FUNCTION_BLOCK FD_ConvoyerDevice EXTENDS FD_Device IMPLEMENTS ITF_Convoyer
VAR_INPUT
END_VAR

VAR_OUTPUT
END_VAR

VAR 
	//===================== Variable
	eSource 						 : E_Convoyer;
  eDestination 				 : E_Convoyer;
	
	bRouteRequest				 : BOOL;
	bCarrierWaiting   	 : BOOL;
	bRouteGranted 			 : BOOL;
	
	bTranspOutRequest    : BOOL;
	bTranspOutBusy       : BOOL;
	bTranspOutDone       : BOOL;
	
	//===================== Instance
	fbStopperCarrieConvoyer						: FB_PneuCyl_Stopper  (GVL_Customer.C_Name_StopperCarrieConvoyer,
																													GVL_Customer.C_ID_StopperCarrieConvoyer
																										  		);																												
																												
	fbMotorConvoyer										: FB_SimpleMotor      (GVL_Customer.C_Name_ConvoyerDcMotor,
																													 GVL_Customer.C_ID_MotorComvoyer
																										  		);
																													
	fbReadHead												: FB_ReadHead        	(GVL_Customer.C_Name_ReadHead,
																													GVL_Customer.C_ID_ReadHead
																										  		); 
																													
END_VAR

VAR CONSTANT
	// --------------------------Base------------------
	C_SeqStep_OnBasePos_Start															: UINT :=  1; 
	C_SeqStep_OnBasePos_WaitOpMode												: UINT :=  2;
	C_SeqStep_OnBasePos_Done															: UINT :=  30; 
	
	// --------------------------Auto Sequence------------------
	C_SeqStep_Auto_Start																	: UINT :=  10;
	C_SeqStep_Auto_Wait_Carrier_At_Stopper								: UINT :=  110;
	C_SeqStep_Auto_Read_Destination_Once									: UINT :=  120;
	C_SeqStep_Auto_Ask_RouteManager_For_A_Route						: UINT :=  130;
	C_SeqStep_Auto_Inject_Carrier_IntoGranted_Route				: UINT :=  140;
	C_SeqStep_Auto_End																		: UINT :=  150;
	
END_VAR


//******* Important and necessary
SUPER^();  
//====================================
IF NOT Enable THEN RETURN; END_IF

fbStopperCarrieConvoyer();
fbMotorConvoyer();
fbReadHead();

PROPERTY CarrierWaiting : BOOL
GET
CarrierWaiting := bCarrierWaiting;
END_GET
SET
bCarrierWaiting := CarrierWaiting;
END_SET
END_PROPERTY

PROPERTY Destination : E_Convoyer
GET
Destination := eDestination;
END_GET
SET
eDestination := Destination;
END_SET
END_PROPERTY

//FB_Init ist immer implizit verfügbar und wird primär für die Initialisierung verwendet.
//Der Rückgabewert wird nicht ausgewertet. Für gezielte Einflussnahme können Sie
//die Methoden explizit deklarieren und darin mit dem Standard-Initialisierungscode 
//zusätzlichen Code bereitstellen. Sie können den Rückgabewert auswerten.
METHOD FB_Init: BOOL
VAR_INPUT    
	bInitRetains					: BOOL; 					// TRUE: Die Retain-Variablen werden initialisiert (Reset warm / Reset kalt)    
	bInCopyCode						: BOOL;  					// TRUE: Die Instanz wird danach in den Kopiercode kopiert (Online-Change)
	
	I_Name                : STRING;         //  Name
	I_ID                  : UINT;           // ID
  I_itfOwner					  : ITF_Owner;      // owner 
END_VAR
END_METHOD

METHOD mAutomatic : E_CmdState
VAR_INPUT
	I_bExecute	: BOOL;
END_VAR

SUPER^.mAutomatic(TRUE);
END_METHOD

METHOD mCmdExec_Auto : E_CmdState
VAR_INPUT
END_VAR

VAR
    L_eCmd 			: E_CmdState;
END_VAR

CASE SequenceID OF

  //******************************************************* Idle 
  C_SeqStep_Idle: 
  	SequenceID       :=  C_SeqStep_Start;
  
  //****************************************************** Start
  C_SeqStep_Start:
		bRouteRequest 			:= FALSE;
    bRouteGranted 			:= FALSE;
    bTranspOutRequest 	:= FALSE;
    bTranspOutDone 			:= FALSE; 	
  	SequenceID          := C_SeqStep_Auto_Wait_Carrier_At_Stopper;
		
	C_SeqStep_Auto_Wait_Carrier_At_Stopper :
	
	IF fbStopperCarrieConvoyer.CarriePresent 
		THEN
      SequenceID := C_SeqStep_Auto_Read_Destination_Once;
  END_IF
	
	C_SeqStep_Auto_Read_Destination_Once:
	// Read destination one.
  	IF fbReadHead.mRead(TRUE) = E_CmdState.Succeeded 
			THEN
  	    eDestination 		:= fbReadHead.ReadDestination;
  	    SequenceID 			:= C_SeqStep_Auto_Ask_RouteManager_For_A_Route;
  	END_IF
	
	C_SeqStep_Auto_Ask_RouteManager_For_A_Route:
	// Ask RouteManager for a route.
 		bRouteRequest := TRUE;
		
    IF bRouteGranted 
			THEN
    		bTranspOutRequest  := TRUE;
    	  SequenceID         := C_SeqStep_Auto_Inject_Carrier_IntoGranted_Route;
    	END_IF

	 C_SeqStep_Auto_Inject_Carrier_IntoGranted_Route:
      // Inject carrier into granted route.				
		IF mCmdExec_TranspOut(bTranspOutRequest ) = E_CmdState.Succeeded 
			THEN
      	bRouteRequest     := FALSE;
      	bRouteGranted     := FALSE;
      	bTranspOutRequest := FALSE;
      	SequenceID        := C_SeqStep_Auto_End;
     END_IF
									
  C_SeqStep_Error: 
    //************* all FB reset
 
 	C_SeqStep_Auto_End:
	  //**********************End 
		SequenceID := C_SeqStep_Start;
  		
END_CASE
END_METHOD

METHOD mCmdExec_BasePos : E_CmdState
VAR_INPUT
END_VAR

CASE SequenceID OF
  //******************************************************* Idle 
  C_SeqStep_Idle: 
  	;
  //****************************************************** Start
  C_SeqStep_OnBasePos_Start:
	// Home position for LTU is MIDDLE.
		fbMotorConvoyer.mStopMotor(TRUE);
		IF E_CmdState.Succeeded  = fbStopperCarrieConvoyer.mCallBase(TRUE)
			THEN
				Homed := TRUE;
  	  	Ready := TRUE;
  	  	SequenceID := C_SeqStep_OnBasePos_Done;
		END_IF
		
  C_SeqStep_Error: 
    //************* all FB reset
    mCmdExec_BasePos := mDone(); 
  //**********************Done
 	C_SeqStep_OnBasePos_Done:
  	mCmdExec_BasePos := mDone();
END_CASE
END_METHOD

METHOD mCmdExec_Service : E_CmdState
VAR_INPUT
END_VAR
;
END_METHOD

METHOD mCmdExec_TranspOut : E_CmdState
VAR_INPUT
	I_bExecute 			: BOOL;
END_VAR

IF NOT I_bExecute 
	THEN
    bTranspOutBusy := FALSE;
    mCmdExec_TranspOut := E_CmdState.Idle;
    RETURN;
END_IF

// Route not granted yet.
// Route noch nicht freigegeben
IF NOT bRouteGranted 
	THEN
  	mCmdExec_TranspOut := E_CmdState.NotReady;
    RETURN;
END_IF

bTranspOutBusy := TRUE;
bTranspOutDone := FALSE;

// Open stopper: stopper down = carrier can pass.
fbStopperCarrieConvoyer.mCallWork(TRUE);

// Start conveyor motor.
fbMotorConvoyer.mStartMotor(TRUE);

// Wait until carrier leaves stopper sensor.
IF NOT fbStopperCarrieConvoyer.CarriePresent 
	THEN
  	// Stop local injection.
  	fbMotorConvoyer.mStopMotor(TRUE);
		
  	// Close stopper again.
  	fbStopperCarrieConvoyer.mCallBase(TRUE);
  	bTranspOutBusy := FALSE;
  	bTranspOutDone := TRUE;
  	mCmdExec_TranspOut := E_CmdState.Succeeded;
  	RETURN;
END_IF
END_METHOD

METHOD mHold : E_CmdState
VAR_INPUT
	I_bExecute	: BOOL;
END_VAR
END_METHOD

METHOD mHome : E_CmdState
VAR_INPUT
	I_bExecute	: BOOL;
END_VAR
SUPER^.mHome(I_bExecute);
END_METHOD

METHOD mRelease : E_CmdState
VAR_INPUT
	I_bExecute	: BOOL;
END_VAR
END_METHOD

METHOD mSequence : E_CmdState
VAR_INPUT
	I_bExecute				: BOOL;
END_VAR

VAR
	L_eState 					: E_CmdState;
END_VAR
mSequence := SUPER^.mSequence(I_bExecute);	


// Generic checks from parent
L_eState := SUPER^.mSequence(I_bExecute := I_bExecute);

IF L_eState <> E_CmdState.Busy 
	THEN
    mSequence := L_eState;
    RETURN;
END_IF

CASE Mode OF
	E_Mode.Homing:
		mSequence := mCmdExec_BasePos();
	E_Mode.Auto:
		mSequence := mCmdExec_Auto();
	E_Mode.Service:
		mSequence := mCmdExec_Service();	
END_CASE
END_METHOD

METHOD mService : E_CmdState
VAR_INPUT
	I_bExecute	: BOOL;
END_VAR
END_METHOD

METHOD mStop : E_CmdState
VAR_INPUT
	I_bExecute	: BOOL;
END_VAR
END_METHOD

PROPERTY RouteGranted : BOOL
GET
RouteGranted := bRouteGranted;
END_GET
SET
bRouteGranted := RouteGranted;
END_SET
END_PROPERTY

PROPERTY RouteRequest : BOOL
GET
RouteRequest := bRouteRequest;
END_GET
SET
bRouteRequest := RouteRequest;
END_SET
END_PROPERTY

PROPERTY Source : E_Convoyer
GET
Source := eSource;
END_GET
SET
eSource := Source;
END_SET
END_PROPERTY

PROPERTY TranspOutBusy : BOOL
GET
TranspOutBusy := bTranspOutBusy;
END_GET
SET
bTranspOutBusy := TranspOutBusy;
END_SET
END_PROPERTY

PROPERTY TranspOutDone : BOOL
GET
TranspOutDone := bTranspOutDone;
END_GET
SET
bTranspOutDone := TranspOutDone;
END_SET
END_PROPERTY

PROPERTY TranspOutRequest : BOOL
GET
TranspOutRequest := bTranspOutRequest;
END_GET
SET
bTranspOutRequest := TranspOutRequest;
END_SET
END_PROPERTY

END_FUNCTION_BLOCK

(* stored: Version 1.1.0.1, ProductVersion 3.1.4026.18
   POU FD_ConvoyerDevice: Id {f58c6f5d-3b14-41fa-923e-c299a6fe3b56}, SpecialFunc None
   Folder 01 Properties: Id {cd138be3-3b0b-4a38-a306-c41018d06bbb}
   Folder 02 Methodes: Id {6037a7d3-2441-4a02-b758-7b67f5b9751c}
   Folder 100 CmdExecute: Id {915cb2b9-e0a9-4914-87d5-0baeeaed19ff}
   Folder 400 Fx: Id {777dcdf1-ad3f-4720-8084-0c004ef66f79}
   Property CarrierWaiting: Id {05c90862-a01c-4d41-bb8b-9f422f1fc899}
   Get Get: Id {67938f79-f29a-4cbe-8d7d-487753b2d290}
   Set Set: Id {9e15df62-c638-412d-b1f4-b4bf0ee0e80d}
   Property Destination: Id {60e01930-c4c2-43cd-a7d9-e5b12f7f1196}
   Get Get: Id {50f207cd-1873-4a37-ac63-f80e4da816e8}
   Set Set: Id {bc36f908-3346-4f37-b28c-03f65b639893}
   Method FB_Init: Id {7868e964-b97f-4b46-9f24-6f16557dff08}
   Method mAutomatic: Id {0e38ef4b-50a5-4c6b-a712-d14a65a1cbe0}
   Method mCmdExec_Auto: Id {973859fe-6ada-4c64-963f-bf319c88cc9e}
   Method mCmdExec_BasePos: Id {eb2de01f-87e9-4e47-9b8c-605e0a054e34}
   Method mCmdExec_Service: Id {d322bdec-4501-4078-818a-8eafd3a95f6f}
   Method mCmdExec_TranspOut: Id {2bdddac8-0ea5-442f-81c6-6021ed68c775}
   Method mHold: Id {46387c63-22e9-4e63-911a-a5aaa6ea0e64}
   Method mHome: Id {0b8d40f6-21bb-47c1-a405-da8066a9c8d8}
   Method mRelease: Id {12251720-22ac-41a7-b04d-07588ae5005c}
   Method mSequence: Id {3b40ca71-71ef-49e1-9faa-1a629e293a02}
   Method mService: Id {11d63726-4dd4-47d5-9688-e549348cfcc2}
   Method mStop: Id {cbc30238-9fbe-4bf6-a78e-b9b20bf3a4ae}
   Property RouteGranted: Id {cd1cb68a-27d6-4b9a-aff7-1fc7113476aa}
   Get Get: Id {d9255acc-bca3-4e38-b863-ea159f4ce6df}
   Set Set: Id {eb76f2eb-5589-4c0e-b893-5d7bf2398402}
   Property RouteRequest: Id {a5fb370a-96f9-4d94-8387-bb7d62846ac8}
   Get Get: Id {a28c8fbe-49de-40da-8e17-df8ad6f76647}
   Set Set: Id {8c120947-2645-4e50-95bc-9fbc28162cae}
   Property Source: Id {6d963e4a-854c-4dd7-91c7-948da36b0f5b}
   Get Get: Id {e71207da-0331-44af-907d-a281da8fb600}
   Set Set: Id {a30af409-5f1c-4e08-b808-7a87cc5aeaca}
   Property TranspOutBusy: Id {b8b5a2ba-94ac-4ae1-b191-a3196eacd9fc}
   Get Get: Id {631c6046-8190-41fd-a8a5-ff75edf18165}
   Set Set: Id {d7fb4dd2-7420-4ae0-ad17-41213018e36d}
   Property TranspOutDone: Id {fa04fbd9-08e0-48f8-9ce8-4fbd3cc4bd4c}
   Get Get: Id {76b7288d-7dee-43b0-a835-8980c9dc7118}
   Set Set: Id {53762087-ce96-4e2c-bc0b-8dfb4b0e588d}
   Property TranspOutRequest: Id {3896cf4c-3a65-4549-83b4-30d9f26b3986}
   Get Get: Id {0477b759-e0c8-4ee6-877e-00686b07c4f1}
   Set Set: Id {f3aacb44-1924-4983-93b4-cfcbe1c746b7} *)
